// TIA Portal project "4063_PLC" (V16)

(* hardware
DEVICE "S71500/ET200MP station_1"  S7-1500 station
   slot 0: "Telaio di montaggio_0"  Rack  6ES7 590-1***0-0AA0
   slot 1: "PLC_4063"  CPU 1511-1 PN  6ES7 511-1AK02-0AB0  V2.8
      slot 3: "Display CPU_1"  6ES7591-1AA00-0AA0
      slot 32768: "Interfaccia PROFINET_1"  X1
         slot 32769: "Porta_1"  X1 P1
         slot 32770: "Porta_2"  X1 P2
      slot 34817: "Virtual CP interface port_1"  Virtual CP interface port  Virtual CP interface port
   slot 2: "DI 16x24VDC HF_1"  DI 16x24VDC HF  6ES7 521-1BH00-0AB0  V2.2
   slot 3: "DQ 16x24VDC/0.5A HF_1"  DQ 16x24VDC/0.5A HF  6ES7 522-1BH01-0AB0  V1.1
   slot 4: "AQ 4xU/I ST_1"  AQ 4xU/I ST  6ES7 532-5HD00-0AB0  V2.2
   slot 5: "DI 16x24VDC HF_2"  DI 16x24VDC HF  6ES7 521-1BH00-0AB0  V2.2
   slot 6: "AQ 2xU/I ST_1"  AQ 2xU/I ST  6ES7 532-5NB00-0AB0  V1.0
   slot 7: "DQ 16x24VDC/0.5A HF_2"  DQ 16x24VDC/0.5A HF  6ES7 522-1BH01-0AB0  V1.1
   slot 8: "DI 16x24VDC HF_3"  DI 16x24VDC HF  6ES7 521-1BH00-0AB0  V2.2
   slot 9: "CP 1542-5_1"  CP 1542-5  6GK7 542-5FX00-0XE0  V2.0
DEVICE "SERVO_11"  GSD.Device
   slot 0: "UR"  Rail
DEVICE "SERVO_1"  GSD.Device
   slot 0: "UR"  Rail
DEVICE "SERVO_2"  GSD.Device
   slot 0: "UR"  Rail
DEVICE "SERVO_3"  GSD.Device
   slot 0: "UR"  Rail
DEVICE "SERVO_4"  GSD.Device
   slot 0: "UR"  Rail
DEVICE "SERVO_5"  GSD.Device
   slot 0: "UR"  Rail
DEVICE "SERVO_6"  GSD.Device
   slot 0: "UR"  Rail
*)

// ===== PLC "PLC_4063"  CPU 1511-1 PN =====

DATA_BLOCK "Data"   // DB1
{ S7_Optimized_Access := 'TRUE' }
VERSION : 0.1
   VAR
      i : Int;
      seed : Int;
      Random_Number_Db : Array[0..1000] of Int;
   END_VAR
BEGIN
END_DATA_BLOCK

FUNCTION_BLOCK "Check_OPCUA_Status"   // FB1, SCL
{ S7_Optimized_Access := 'TRUE' }
VERSION : 0.1
   VAR
      OPC_UA_ServerMethodPre_Instance : OPC_UA_ServerMethodPre;
      OPC_UA_ServerMethodPost_Instance : OPC_UA_ServerMethodPost;
   END_VAR
   VAR_TEMP
      Done_Server_OPCUA : Bool;
      Busy_Server_OPCUA : Bool;
      Error_Server_OPCUA : Bool;
      Status_Server_OPCUA : DWord;
      UAMethod_Called : Bool;
      UAMethod_InParameters : Int;
      Check_Status : Bool;
      UAMethod_Result : DWord;
      UAMethod_Finished : Bool;
      Done_Server_OPCUA_Post : Bool;
      Busy_Server_OPCUA_Post : Bool;
      Error_Server_OPCUA_Post : Bool;
      Status_Server_OPCUA_Post : DWord;
      UAMethod_OutParameters : Int;
   END_VAR
BEGIN
   #Check_Status := FALSE;


   WHILE #Check_Status DO

       #OPC_UA_ServerMethodPre_Instance(
                                        Done => #Done_Server_OPCUA,
                                        Busy => #Busy_Server_OPCUA,
                                        Error => #Error_Server_OPCUA,
                                        Status => #Status_Server_OPCUA,
                                        UAMethod_Called => #UAMethod_Called,
                                        UAMethod_InParameters := #UAMethod_InParameters
       );
       #OPC_UA_ServerMethodPost_Instance(
                                         UAMethod_Result := #UAMethod_Result,
                                         UAMethod_Finished := #UAMethod_Finished,
                                         Done => #Done_Server_OPCUA_Post,
                                         Busy => #Busy_Server_OPCUA_Post,
                                         Error => #Error_Server_OPCUA_Post,
                                         Status => #Status_Server_OPCUA_Post,
                                         UAMethod_OutParameters := #UAMethod_OutParameters
       );


   END_WHILE;
END_FUNCTION_BLOCK

FUNCTION "Pseudo_Random_Number" : Void   // FC1, SCL
{ S7_Optimized_Access := 'TRUE' }
VERSION : 0.1
   VAR_INPUT
      leng_array : Int;
   END_VAR
   VAR_TEMP
      i : Int;
      Seed : Int;
   END_VAR
BEGIN
   // index Identifier while looping 
   "Data".i := 0;

   //Random seed 
   "Data".seed := 10;

   // Create and append random nuber to an Array 
   WHILE #leng_array > "Data".i DO

       "Data".seed := "Data".seed + "Data".i;
       "Data".i := "Data".i + 1;

       "Data".Random_Number_Db["Data".i] := "Data".seed ;

   END_WHILE;
END_FUNCTION

ORGANIZATION_BLOCK "Main"   // OB1, LAD, ProgramCycle
TITLE = "Main Program Sweep (Cycle)"
{ S7_Optimized_Access := 'TRUE' }
VERSION : 0.1
   VAR_INPUT
      Initial_Call : Bool;   // Initial call of this OB
      Remanence : Bool;   // =True, if remanent data are available
   END_VAR
   VAR_TEMP
      Random_Number : Array[0..100] of Int;
   END_VAR
BEGIN

REGION Network 1 (STL)
         CALL  "Pseudo_Random_Number"
         ( leng_array := 50
         );
END_REGION
END_ORGANIZATION_BLOCK